Fanuc TP program (LS listing): CELL_IN.LS

/PROG  CELL_IN
/ATTR
OWNER		= MNEDITOR;
COMMENT		= "stub: entry into the drawing area";
PROG_SIZE	= 0;
CREATE		= DATE 26-09-08  TIME 12:00:00;
MODIFIED	= DATE 26-09-08  TIME 12:00:00;
FILE_NAME	= ;
VERSION		= 0;
LINE_COUNT	= 3;
MEMORY_SIZE	= 0;
PROTECT		= READ_WRITE;
TCD:  STACK_SIZE	= 0,
      TASK_PRIORITY	= 50,
      TIME_SLICE	= 0,
      BUSY_LAMP_OFF	= 0,
      ABORT_REQUEST	= 0,
      PAUSE_REQUEST	= 0;
DEFAULT_GROUP	= 1,*,*,*,*;
CONTROL_CODE	= 00000000 00000000;
/MN
   1:  ! CELL_IN stub - replace with a taught ;
   2:  ! approach to the clear plane on the real cell ;
   3:  UFRAME_NUM=1 ;
/POS
/END
